FUNCTION_BLOCK QueryInterfaceResettables IMPLEMENTS I_ComponentVisitor
VAR
	Reset	   : ARRAY[0..10] OF I_Resettable;
	ResetCount : DINT;
END_VAR

METHOD GetAllResetComponents
VAR_INPUT
	EntryModule : I_Module;
END_VAR
ResetCount := 0;
EntryModule.Components.Accept(THIS^);
END_METHOD

METHOD VisitComponent
VAR_INPUT
	Component : I_Component;
END_VAR
IF __QUERYINTERFACE(Component, Reset[ResetCount]) THEN
	ResetCount := ResetCount + 1;
END_IF
END_METHOD

END_FUNCTION_BLOCK

(* stored: Version 1.1.0.1, ProductVersion 3.1.4026.18
   POU QueryInterfaceResettables: Id {e97e9586-170d-4915-83da-922890bb21c7}, SpecialFunc None
   Method GetAllResetComponents: Id {89dce528-9d78-41f2-89b1-208848a91f23}
   Method VisitComponent: Id {d878cc57-b009-4d19-a6c0-efec38d1962d} *)
